TYPE s_DaraSampleSetQty :
STRUCT
	nonDefectiveQty : INT;
	defectiveQty	:INT;
END_STRUCT
END_TYPE

(* stored: Version 1.1.0.1, ProductVersion 3.1.4024.11
   DUT s_DaraSampleSetQty: Id {d4d4d2d4-5476-4f68-bdba-015d3852f052} *)
